TEXTLIST CycleType
  0 = ' '
  1 = 'Continuous Cycle'
  2 = 'Single Cycle'
  3 = 'other state'
   = ''
END_TEXTLIST

(* stored: Version 1.1.0.1, ProductVersion 3.1.4024.12
   TextList CycleType: Id {50519c34-b1da-4461-9772-cc7ecae3996d} *)
